(* PLC project PLC411_MAIN, home PLC411_MAIN 1 *)
(* stored: creationDateTime 2019-11-13T09:37:45, productRelease 0, modificationDateTime 2023-05-04T09:24:28, version 0 *)

(* Increment of source value *)
FUNCTION Inc : INT
  VAR_INPUT
    IN : BOOL;  (* execution allow *)
    V : INT;  (* source value *)
  END_VAR
  VAR
    Val : INT;
  END_VAR

            Val:= V;

IF IN = TRUE THEN
  Val:= V+1;
END_IF;

Inc:= Val;


          
END_FUNCTION

(* Decrement of source value *)
FUNCTION Dec : INT
  VAR_INPUT
    IN : BOOL;  (* execution allow *)
    V : INT;  (* source value *)
  END_VAR
  VAR
    Val : INT;
  END_VAR

            Val:= V;

IF IN = TRUE AND Val > 0 THEN
  Val:= V-1;
END_IF;

Dec:= Val;


          
END_FUNCTION

(* Increment of source value (limited) *)
FUNCTION IncLim : INT
  VAR_INPUT
    IN : BOOL;  (* execution allow *)
    V : INT;  (* value *)
    Mn : INT;  (* minimum *)
    Mx : INT;  (* maximum *)
  END_VAR
  VAR
    Val : INT;
  END_VAR

            Val:= Inc(IN:=IN, V:=V);
Val:= LIMIT(MN:=Mn, IN:=Val, MX:=Mx);
IncLim:= Val;
          
END_FUNCTION

(* Decrement of source value (limited) *)
FUNCTION DecLim : INT
  VAR_INPUT
    IN : BOOL;  (* execution allow *)
    V : INT;  (* value *)
    Mn : INT;  (* minimum *)
    Mx : INT;  (* maximum *)
  END_VAR
  VAR
    Val : INT;
  END_VAR

            Val:= Dec(IN:=IN, V:=V);
Val:= LIMIT(MN:=Mn, IN:=Val, MX:=Mx);
DecLim:= Val;
          
END_FUNCTION

(* RAMP-signal (from 0 to 1000) *)
FUNCTION Ramp1000 : WORD
  VAR_INPUT
    IN : BOOL;  (* execution allow *)
    V : WORD;  (* previous RAMP-signal *)
  END_VAR
  VAR
    Val : INT;
  END_VAR

            Val:= WORD_TO_INT(V);

IF IN = TRUE THEN

  Val:= Val+1;
  IF Val >= 1000 THEN
    Val:= 0;
  END_IF;

END_IF;

Ramp1000:= INT_TO_WORD(Val);


          
END_FUNCTION

(* Set bit value in source word *)
FUNCTION SetBitWo : WORD
  VAR_INPUT
    Wo : WORD := 0;  (* source word *)
    Pos : BYTE := 0;  (* bit position (0..15) *)
    Val : BOOL := FALSE;  (* bit value *)
  END_VAR
  VAR
    Mask : WORD := 0;
  END_VAR

            Mask:= REAL_TO_WORD(EXPT(INT_TO_REAL(2),BYTE_TO_INT(Pos)));
IF Val = FALSE THEN
  SetBitWo:= (Wo AND NOT(Mask));
ELSE
  SetBitWo:= (Wo OR Mask);
END_IF;
          
END_FUNCTION

(* 16-bit coder *)
FUNCTION Cd16 : WORD
  VAR_INPUT
    In0 : BOOL := FALSE;  (* value of 0-bit *)
    In1 : BOOL := FALSE;  (* value of 1-bit *)
    In2 : BOOL := FALSE;  (* value of 2-bit *)
    In3 : BOOL := FALSE;  (* value of 3-bit *)
    In4 : BOOL := FALSE;  (* value of 4-bit *)
    In5 : BOOL := FALSE;  (* value of 5-bit *)
    In6 : BOOL := FALSE;  (* value of 6-bit *)
    In7 : BOOL := FALSE;  (* value of 7-bit *)
    In8 : BOOL := FALSE;  (* value of 8-bit *)
    In9 : BOOL := FALSE;  (* value of 9-bit *)
    In10 : BOOL := FALSE;  (* value of 10-bit *)
    In11 : BOOL := FALSE;  (* value of 11-bit *)
    In12 : BOOL := FALSE;  (* value of 12-bit *)
    In13 : BOOL := FALSE;  (* value of 13-bit *)
    In14 : BOOL := FALSE;  (* value of 14-bit *)
    In15 : BOOL := FALSE;  (* value of 15-bit *)
  END_VAR
  VAR
    Val : WORD := 0;
  END_VAR

            Val:= SetBitWo(Wo:=Val, Pos:=INT_TO_BYTE(0), Val:=In0);
Val:= SetBitWo(Wo:=Val, Pos:=INT_TO_BYTE(1), Val:=In1);
Val:= SetBitWo(Wo:=Val, Pos:=INT_TO_BYTE(2), Val:=In2);
Val:= SetBitWo(Wo:=Val, Pos:=INT_TO_BYTE(3), Val:=In3);
Val:= SetBitWo(Wo:=Val, Pos:=INT_TO_BYTE(4), Val:=In4);
Val:= SetBitWo(Wo:=Val, Pos:=INT_TO_BYTE(5), Val:=In5);
Val:= SetBitWo(Wo:=Val, Pos:=INT_TO_BYTE(6), Val:=In6);
Val:= SetBitWo(Wo:=Val, Pos:=INT_TO_BYTE(7), Val:=In7);
Val:= SetBitWo(Wo:=Val, Pos:=INT_TO_BYTE(8), Val:=In8);
Val:= SetBitWo(Wo:=Val, Pos:=INT_TO_BYTE(9), Val:=In9);
Val:= SetBitWo(Wo:=Val, Pos:=INT_TO_BYTE(10), Val:=In10);
Val:= SetBitWo(Wo:=Val, Pos:=INT_TO_BYTE(11), Val:=In11);
Val:= SetBitWo(Wo:=Val, Pos:=INT_TO_BYTE(12), Val:=In12);
Val:= SetBitWo(Wo:=Val, Pos:=INT_TO_BYTE(13), Val:=In13);
Val:= SetBitWo(Wo:=Val, Pos:=INT_TO_BYTE(14), Val:=In14);
Val:= SetBitWo(Wo:=Val, Pos:=INT_TO_BYTE(15), Val:=In15);
Cd16:= Val;

          
END_FUNCTION

(* Get bit value from source word *)
FUNCTION GetBitWo : BOOL
  VAR_INPUT
    Wo : WORD := 0;  (* source word *)
    Pos : BYTE := 0;  (* bit position (0..15) *)
  END_VAR
  VAR
    Mask : WORD := 0;
  END_VAR

            Mask:= REAL_TO_WORD(EXPT(INT_TO_REAL(2),BYTE_TO_INT(Pos)));
GetBitWo:= ((Wo AND Mask) > 0);

          
END_FUNCTION

(* Calculate scale angle factor *)
FUNCTION ScaleA_Ka : REAL
  VAR_INPUT
    Ex : BOOL := FALSE;  (* execution allow *)
    V1 : REAL := 0.0;  (* value of low point *)
    V2 : REAL := 0.0;  (* value of high point *)
    Y1 : REAL := 0.0;  (* calibration value of low point *)
    Y2 : REAL := 0.0;  (* calibration value of high point *)
    Ka : REAL := 0.0;  (* source value of the factor *)
  END_VAR

            IF Ex = TRUE THEN
  ScaleA_Ka:= (Y2-Y1)/(V2-V1);
ELSE  
  ScaleA_Ka:= Ka;
END_IF;

          
END_FUNCTION

(* Calculate scale offset factor *)
FUNCTION ScaleA_Kb : REAL
  VAR_INPUT
    Ex : BOOL := FALSE;  (* execution allow *)
    V1 : REAL := 0.0;  (* value of low point *)
    V2 : REAL := 0.0;  (* value of high point *)
    Y1 : REAL := 0.0;  (* calibration value of low point *)
    Y2 : REAL := 0.0;  (* calibration value of high point *)
    Kb : REAL := 0.0;  (* source value of the factor *)
  END_VAR

            IF Ex = TRUE THEN
  ScaleA_Kb:= ((Y1*V2)-(Y2*V1))/(V2-V1);
ELSE  
  ScaleA_Kb:= Kb;
END_IF;

          
END_FUNCTION

(* Scale of analog value *)
FUNCTION ScaleA : REAL
  VAR_INPUT
    Ex : BOOL := FALSE;  (* execution allow *)
    V : REAL := 0.0;  (* value of curent point *)
    Ka : REAL := 0.0;  (* angle factor *)
    Kb : REAL := 0.0;  (* offset factor *)
    Y : REAL := 0.0;  (* source scale value *)
  END_VAR

            IF Ex = TRUE THEN
  ScaleA:= (Ka*V)+Kb;
ELSE  
  ScaleA:= Y;
END_IF;

          
END_FUNCTION

(* TON Periodical Blink *)
FUNCTION_BLOCK TONb
  VAR_INPUT
    IN : BOOL := FALSE;  (* TON.Start/Stop *)
    PT : TIME := T#0ms;  (* TON.Period *)
  END_VAR
  VAR_OUTPUT
    Q : BOOL := FALSE;  (* TON.BlinkQuit (period for Q = FALSE, pediod for Q=TRUE) *)
    ET : TIME := T#0ms;  (* TON.EstimatedTime *)
  END_VAR
  VAR
    TON0 : TON;
    TON1 : TON;
  END_VAR

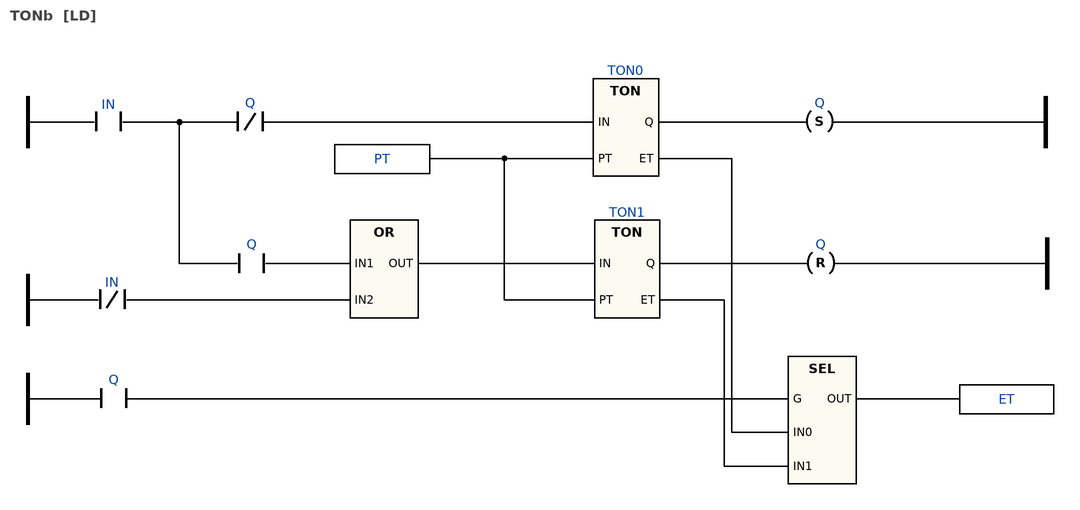
(* LD diagram, written out as Structured Text *)
TON0(IN := IN AND NOT Q, PT := PT);
IF TON0.Q THEN Q := TRUE; END_IF;
TON1(IN := IN AND Q OR NOT IN, PT := PT);
IF TON1.Q THEN Q := FALSE; END_IF;
ET := SEL(Q, TON0.ET, TON1.ET);
END_FUNCTION_BLOCK

(* TON Continuous *)
FUNCTION_BLOCK TONc
  VAR_INPUT
    IN : BOOL := FALSE;  (* start command *)
  END_VAR
  VAR_OUTPUT
    Q : BOOL := FALSE;  (* status *)
    ET : TIME := T#0ms;  (* estimated time *)
  END_VAR
  VAR
    TON1 : TON;
    TON1_IN : BOOL := FALSE;
    TON1_TM : TIME := T#600000ms;
    TON1Inc : TON;
    TON1Inc_IN : BOOL := FALSE;
    TON1Inc_TM : TIME := T#300000ms;
  END_VAR

            TON1_IN   := IN;
TON1Inc_IN:= IN;

IF TON1Inc.Q = TRUE THEN
  TON1_TM   := ADD_TIME(IN1:=TON1_TM, IN2:=TON1Inc_TM);
  TON1Inc_IN:= FALSE;
END_IF;

TON1(IN:=TON1_IN, PT:=TON1_TM);
TON1Inc(IN:=TON1Inc_IN, PT:=TON1Inc_TM);

Q := TON1.Q;
ET:= TON1.ET;

          
END_FUNCTION_BLOCK

(* TON msec *)
FUNCTION_BLOCK TONms
  VAR_INPUT
    IN : BOOL := FALSE;  (* TON.Start/Stop *)
    MS : DWORD := 0;  (* TON.Period (msec) *)
  END_VAR
  VAR_OUTPUT
    Q : BOOL := FALSE;  (* TON.Status (FALSE - counting, TRUE - done) *)
    ET : TIME := T#0ms;  (* TON.EstimatedTime *)
    ETMS : DWORD := 0;  (* TON.EstimatedTime (ms) *)
  END_VAR
  VAR
    TON1 : TON;
    TON1_TM : TIME := T#0ms;
  END_VAR

            IF IN = TRUE THEN
  
  IF MS > 0 THEN
    TON1_TM:= REAL_TO_TIME(DWORD_TO_REAL(MS)/1000.0);
  END_IF;
  
END_IF;

TON1(IN:=IN, PT:=TON1_TM);

IF (MS > 0 AND TON1.Q = TRUE) OR (MS = 0) THEN
  Q:= TRUE;
ELSE
  Q:= FALSE;
END_IF;

ET:= TON1.ET;
ETMS:= REAL_TO_DWORD(TIME_TO_REAL(TON1.ET)*1000.0);

          
END_FUNCTION_BLOCK

(* TON sec *)
FUNCTION_BLOCK TONs
  VAR_INPUT
    IN : BOOL := FALSE;  (* TON.Start/Stop *)
    SEC : WORD := 0;  (* TON.Period (sec) *)
  END_VAR
  VAR_OUTPUT
    Q : BOOL := FALSE;  (* TON.Status (FALSE - counting, TRUE - done) *)
    ET : TIME := T#0ms;  (* TON.EstimatedTime *)
    ETMS : DWORD := 0;  (* TON.EstimatedTime (ms) *)
  END_VAR
  VAR
    TON1 : TON;
    TON1_TM : TIME := T#0ms;
  END_VAR

            IF IN = TRUE THEN
  
  IF SEC > 0 THEN
    TON1_TM:= REAL_TO_TIME(WORD_TO_REAL(SEC));
  END_IF;
  
END_IF;

TON1(IN:=IN, PT:=TON1_TM);

IF (SEC > 0 AND TON1.Q = TRUE) OR (SEC = 0) THEN
  Q:= TRUE;
ELSE
  Q:= FALSE;
END_IF;

ET:= TON1.ET;
ETMS:= REAL_TO_DWORD(TIME_TO_REAL(TON1.ET)*1000.0);

          
END_FUNCTION_BLOCK

(* Filtration of discrete value *)
FUNCTION_BLOCK FiltrD
  VAR_INPUT
    Ex : BOOL := FALSE;  (* execution allow *)
    V : BOOL := FALSE;  (* source value *)
    Tm : TIME := T#0ms;  (* filter delay (ms) *)
  END_VAR
  VAR_OUTPUT
    Ov : BOOL := FALSE;  (* filtered source value *)
  END_VAR
  VAR
    Val : BOOL := FALSE;
    TON0 : TON;
    TON1 : TON;
  END_VAR

            TON0(IN:=AND(Ex, NOT(V)), PT:=Tm);
TON1(IN:=AND(Ex, V), PT:=Tm);

IF TON0.Q = TRUE THEN
  Val:= FALSE;
END_IF;

IF TON1.Q = TRUE THEN
  Val:= TRUE;
END_IF;

Ov:= Val;

          
END_FUNCTION_BLOCK

(* Filtration of analog value *)
FUNCTION_BLOCK FiltrA
  VAR_INPUT
    Ex : BOOL := FALSE;  (* execution allow *)
    V : REAL := 0.0;  (* source value *)
    K : REAL := 0.0;  (* filter factor (0.0 .. 1.0) *)
  END_VAR
  VAR_OUTPUT
    Ov : REAL := 0.0;  (* filtered source value *)
  END_VAR
  VAR
    Val : REAL := 0.0;  (* stored value *)
    Klim : REAL := 0.0;  (* stored value *)
  END_VAR

            IF Ex = TRUE THEN
  Klim:= LIMIT(MN:=0.0, IN:=K, MX:=1.0);
  Val := (Klim*V)+(1.0-Klim)*Ov;
ELSE
  Val:= V;
END_IF;

Ov:= Val;

          
END_FUNCTION_BLOCK

(* 2-Position Regulator *)
FUNCTION_BLOCK Reg2p
  VAR_INPUT
    IN : BOOL := FALSE;  (* Regulator.Start/Stop *)
    V : REAL := 0.0;  (* Process Value *)
    Sp : REAL := 0.0;  (* Setpoint *)
    Hy : REAL := 0.0;  (* Hysteresis (+/- from Sp) for Q.On/Off *)
    Tm : TIME := T#0ms;  (* Output delay *)
  END_VAR
  VAR_OUTPUT
    Q : BOOL := FALSE;  (* Output command *)
  END_VAR
  VAR
    First : BOOL := FALSE;  (* First iteration is completed (TRUE) *)
    TON1 : TON;
    TON1_IN : BOOL := FALSE;
  END_VAR

            IF IN = TRUE THEN
  
  IF (V < Sp AND First = FALSE) OR (V < (Sp-Hy)) THEN
    TON1_IN:= TRUE;
  ELSIF (V > (Sp+Hy)) THEN
    TON1_IN:= FALSE;
  END_IF;

  IF First = FALSE THEN
    First:= TRUE;
  END_IF;
  
ELSE
  First:= FALSE;
  TON1_IN:= FALSE;
  Q:= FALSE;
END_IF;

Q:= TON1.Q;

TON1(IN:=TON1_IN, PT:=Tm);

          
END_FUNCTION_BLOCK

(* Diagnostic of the Control Loop *)
FUNCTION_BLOCK LoopCtrl
  VAR_INPUT
    V : REAL := 0.0;  (* Process Value *)
    CHi : BOOL := FALSE;  (* HighAlarmZone.Allow *)
    DHi : REAL := 0.0;  (* HighAlarmZone.Setpoint *)
    THi : TIME := T#0ms;  (* HighAlarmZone.Delay *)
    CLo : BOOL := FALSE;  (* LowAlarmZone.Allow *)
    DLo : REAL := 0.0;  (* LowAlarmZone.Setpoint *)
    TLo : TIME := T#0ms;  (* LowAlarmZone.Delay *)
  END_VAR
  VAR_OUTPUT
    Q : BOOL := FALSE;  (* Result (TRUE - no breakage, FALSE - breakage) *)
    OK : BYTE := 0;  (* Result code (0 - no breakage, 1 - breakage in Low Zone, 2 - breakage in High Zone) *)
  END_VAR
  VAR
    TON1 : TON;
    TON1_IN : BOOL := FALSE;
    TON1_PT : TIME := T#0ms;
    K : BYTE := 0;  (* Result code (local) *)
  END_VAR

            IF (V < DLo AND CLo = TRUE) THEN
  K:= 1;
  TON1_PT:= TLo;
ELSIF (V > DHi AND CHi = TRUE) THEN
  K:= 2;
  TON1_PT:= THi;
ELSE
  K:= 0;
END_IF;

IF K > 0 THEN
  TON1_IN:= TRUE;
  IF TON1.Q = TRUE THEN
    OK:= K;
  END_IF;
ELSE
  TON1_IN:= FALSE;
  OK:= 0;
END_IF;

TON1(IN:=TON1_IN, PT:=TON1_PT);

IF OK > 0 THEN
  Q:= TRUE;
ELSE
  Q:= FALSE;
END_IF;

          
END_FUNCTION_BLOCK

(* PID-controller (v1) *)
FUNCTION_BLOCK PID1
  VAR_INPUT
    Ex : BOOL := FALSE;  (* execution allow *)
    V : REAL := 0.0;  (* source value *)
    Sp : REAL := 0.0;  (* setpoint *)
    Ty : BYTE := 0;  (* type of controller *)
    Pro : BYTE := 0;  (* type of process *)
    Kp : REAL := 0.0;  (* P-factor *)
    Ki : REAL := 0.0;  (* I-factor *)
    Kd : REAL := 0.0;  (* D-factor *)
    Sck : BOOL := FALSE;  (* external command to start regulator cycle *)
    dI : REAL := 0.0;  (* integral zone *)
    dZ : REAL := 0.0;  (* dead zone *)
    Ym : BYTE := 0;  (* type of OY *)
  END_VAR
  VAR_OUTPUT
    Ok : BYTE := 0;  (* result code *)
    OY : REAL := 0.0;  (* regulator value (%) *)
  END_VAR
  VAR
    Er : REAL := 0.0;  (* error delta *)
    ErAbs : REAL := 0.0;  (* error delta (absolute) *)
    ErPrev : REAL := 0.0;  (* error delta (previous cycle) *)
    ErDiff : REAL := 0.0;  (* error delta (diff) *)
    Ppart : REAL := 0.0;  (* P-part *)
    Ipart : REAL := 0.0;  (* I-part *)
    Dpart : REAL := 0.0;  (* D-part *)
    SckSet : BOOL := FALSE;  (* external start (set) *)
    ErrorSet : BOOL := FALSE;  (* e-zone (set) *)
  END_VAR

            (* Ty - regulator type *)
(* = 0 - PID *)
(* = 1 - PI *)
(* = 2 - PD *)
(* = 3 - P *)

(* Pro - process type *)
(* = 0 - increasing (by default) *)
(* = 1 - decreasing *)

(* Ym - type of OY *)
(* = 0 - unipolar    0.0 .. 100.0 % (by default) *)
(* = 1 - bipolar  -100.0 .. 100.0 % *)

(* Ok - result code *)
(* = 0 - work *)
(* = 1 - off *)
(* = 2 - dead (d-)zone *)
(* = 3 - integral (i-)zone *)
(* = 4 - incorrect regulator type *)

(* reset Sck *)
IF Sck = FALSE THEN
  SckSet:= FALSE;
END_IF;

(* test execution allow *)
IF Ex = TRUE THEN
  
  (* test regulator type *)
  IF Ty <= 3 THEN
    
    (* test start *)
    IF Sck = TRUE AND SckSet = FALSE AND ErrorSet = FALSE THEN
      
      SckSet:= TRUE;
      
      (* work *)
      Ok:= 0;
     
      Er    := (Sp-V);
      ErDiff:= (Er-ErPrev);
      ErPrev:= Er;
      ErAbs := ABS(IN:=Er);
      
      (* test d-zone *)
      IF ErAbs >= dZ THEN
        
        (* Ty: 0-PID, 1-PI, 2-PD, 3-P *)
        Ppart:= (Kp*Er);
        
        (* Ty: 0-PID, 1-PI *)
        IF (Ty = 0 OR Ty = 1) AND (ErAbs < dI OR dI = 0.0) AND Ki > 0.0 THEN
          (* i-zone *)
          Ok:= 3;
          Ipart:= (Ipart+Er);
          IF Ipart >= Ki THEN
            Ipart:= Ki;
          END_IF;
          Ipart:= ((1.0/Ki)*Ipart);
        ELSE
          Ipart:= 0.0;
        END_IF;
        
        (*0-PID, 2-PD*)
        IF (Ty = 0 OR Ty = 2) THEN
          Dpart:= (Kd*ErDiff);
        ELSE
          Dpart:= 0.0;
        END_IF;
        
        OY:= (Ppart+Ipart+Dpart)*100.0;
        
      ELSE
        (* d-zone *)
        Ok:= 2;
      END_IF;
      (* end of test d-zone *)
      
    END_IF;
    (* end of test start *)
  
  ELSE
    (* incorrect regulator type *)
    Ok:= 4;
    ErrorSet:= TRUE;
  END_IF;
  (* end of test regulator type *)
  
ELSE
  (* off *)
  Ok:= 1;
END_IF;
(* end of Ex *) 

(* off *)
IF Ok = 1 THEN
  OY       := 0.0;
  SckSet   := FALSE;
  ErrorSet := FALSE;
  Ppart    := 0.0;
  Ipart    := 0.0;
  Dpart    := 0.0;
END_IF;

(* error of regulator type *)
IF ErrorSet = TRUE THEN
  OY       := 0.0;
END_IF;

(* scale OY by type of process *)
IF Pro = 1 THEN
  (* decreasing *)
  OY:= (100.0-OY);
END_IF;

(* scale OY by type of output *)
IF Ym = 1 THEN
  (* bipolar *)
  OY:= LIMIT(MN:=-100.0, IN:=OY, MX:=100.0);
ELSE
  (* unipolar *)
  OY:= LIMIT(MN:=0.0, IN:=OY, MX:=100.0);
END_IF;

          
END_FUNCTION_BLOCK

(* PID-controller (v2) *)
FUNCTION_BLOCK PID2
  VAR_INPUT
    Ex : BOOL := FALSE;  (* execution allow *)
    V : REAL := 0.0;  (* source value *)
    Sp : REAL := 0.0;  (* setpoint *)
    Ty : BYTE := 0;  (* type of controller *)
    Pro : BYTE := 0;  (* type of process *)
    Kp : REAL := 0.0;  (* P-factor *)
    Ki : REAL := 0.0;  (* I-factor *)
    Kd : REAL := 0.0;  (* D-factor *)
    Tm : DWORD := 1000;  (* cycle time (ms) *)
    dI : REAL := 0.0;  (* integral zone *)
    dZ : REAL := 0.0;  (* dead zone *)
    Ym : BYTE := 0;  (* type of OY *)
  END_VAR
  VAR_OUTPUT
    Ok : BYTE := 0;  (* result code *)
    OY : REAL := 0.0;  (* regulator value (%) *)
  END_VAR
  VAR
    TON_Work : TON;
    TON_Work_IN : BOOL := FALSE;
    TON_Work_TM : TIME := T#0ms;
    PID1_1 : PID1;
  END_VAR

            PID1_1(Ex:=Ex, V:=V, Sp:=Sp, Ty:=Ty, Pro:=Pro, Kp:=Kp, Ki:=Ki, Kd:=Kd, Sck:=TON_Work.Q, dI:=dI, dZ:=dZ, Ym:=Ym);

Ok:= PID1_1.Ok;
OY:= PID1_1.OY;

IF Ex = TRUE AND Tm > 0 THEN
  TON_Work_TM:= REAL_TO_TIME(DWORD_TO_REAL(Tm)/1000.0);
  TON_Work_IN:= TRUE;
ELSE
  TON_Work_IN:= FALSE;
END_IF;

IF TON_Work.Q = TRUE THEN
  TON_Work_IN:= FALSE;
END_IF;

TON_Work(IN:=TON_Work_IN, PT:=TON_Work_TM);

(* DEBUG *)
(* set Class of debug variables to Output to use its as Outputs of the FB *)
(* set Class of debug variables to Local to hide its *)
(* Deb_P   := PID1_1.Deb_P; *)
(* Deb_I   := PID1_1.Deb_I; *)
(* Deb_D   := PID1_1.Deb_D; *)
(* Deb_Et  := REAL_TO_DWORD(TIME_TO_REAL(TON_Work.ET)*1000.0); *)
(* Deb_dEEt:= PID1_1.Deb_dEEt; *)
(* end of DEBUG *)

          
END_FUNCTION_BLOCK

(* Autotuning of PID-controller *)
FUNCTION_BLOCK PIDtun
  VAR_INPUT
    Ex : BOOL := FALSE;  (* execution allow *)
    V : REAL := 0.0;  (* source value *)
    Diff : REAL := 0.0;  (* difference setpoint *)
    Ty : BYTE := 0;  (* type of controller *)
    Pro : BYTE := 0;  (* type of process *)
  END_VAR
  VAR_OUTPUT
    Ok : BYTE := 0;  (* result code *)
    OY : REAL := 0.0;  (* regulator value *)
    OKp : REAL := 0.0;  (* P-factor *)
    OKi : REAL := 0.0;  (* I-factor *)
    OKd : REAL := 0.0;  (* D-factor *)
    OTm : DWORD := 0;  (* cycle time (ms) *)
  END_VAR
  VAR
    TunDone : BOOL := FALSE;
    Tm1 : REAL := 0.0;  (* t0 (ms) *)
    Tm2 : REAL := 0.0;  (* tu (ms) *)
    TmSum : REAL := 0.0;  (* t (ms) *)
    V1Set : BOOL := FALSE;
    V01 : REAL := 0.0;
    V063 : REAL := 0.0;
    Rr : REAL := 0.0;  (* R *)
    Tm1sec : REAL := 0.0;  (* t0 div 100 *)
    TONcont1 : TONc;
    TONcont1_IN : BOOL := FALSE;
  END_VAR

            (* Ty - regulator type *)
(* = 0 - PID *)
(* = 1 - PI *)
(* = 2 - PD *)
(* = 3 - P *)

(* Pro - process type *)
(* = 0 - increasing (by default) *)
(* = 1 - decreasing *)

(* Ok - result code *)
(* = 0 - work *)
(* = 1 - off *)
(* = 2 - incorrect regulator type *)
(* = 3 - work done success *)

IF Ex = TRUE THEN
  
  IF Ty <= 3 THEN
      
    IF TunDone = FALSE THEN
      
      (* work *)
      Ok:= 0;
      
      IF V1Set = FALSE THEN
        V1Set:= TRUE;
        (* calculate setpoint for V(0.1) by type of process *)
        IF Pro = 1 THEN
          (* decreasing *)
          V01 := (V-(0.1*Diff));
          V063:= (V-(0.63*Diff));
        ELSE
          (* increasing *)
          V01 := (V+(0.1*Diff));
          V063:= (V+(0.63*Diff));
        END_IF;
      END_IF;
      
      (* set Tm1 (ms) *)
      IF V < V01 THEN
        Tm1:= TIME_TO_REAL(TONcont1.ET)*1000.0;
      END_IF;
      
      (* set Tm2 (ms) *)
      IF V >= V063 THEN
        
        TONcont1_IN:= FALSE;
        TunDone    := TRUE;
        
        Tm2   := TIME_TO_REAL(TONcont1.ET)*1000.0;
        TmSum := (Tm1+Tm2);
        OTm   := REAL_TO_DWORD((Tm1*1.875));
        Rr    := (Diff/((TmSum-Tm1)/1000.0));
        Tm1sec:= (Tm1/1000.0);
        (* 1000 - divider to convert msec to sec *)
          
        (* calculate factors by type of regulator *)
        CASE BYTE_TO_INT(Ty) OF
          0:
            (* PID *)
            OKp:= (1.2/(Rr*Tm1sec));
            OKi:= (2.0*Tm1sec);
            OKd:= (0.4*Tm1sec);
          1:
            (* PI *)
            OKp:= (0.8/(Rr*Tm1sec));
            OKi:= (2.0*Tm1sec);
          2:
            (*PD*)
            OKp:= (1.0/(Rr*Tm1sec));
            OKd:= (0.25*Tm1sec);
          3:
            (*P*)
            OKp:= (1.0/(Rr*Tm1sec));
        END_CASE;
        
      END_IF;
      (* end of Tm2 *)
    ELSE
      (* work done success *)
      Ok:= 3;
    END_IF;
    (* end of TunDone *)
  ELSE
    (* incorrect regulator type *)
    Ok:= 2;
  END_IF;
  (* end of Ty *)
ELSE
  (* off *)
  Ok:= 1;
END_IF;
(* end of Ex *)

(* work *)
IF Ok = 0 THEN
  OY         := 100.0;
  TONcont1_IN:= TRUE;
END_IF;

(* off, error *)
IF Ok = 1 OR Ok = 2 THEN
  OY         := 0.0;
  TONcont1_IN:= FALSE;
  V1Set      := FALSE;
  TunDone    := FALSE;
  OKp        := 0.0;
  OKi        := 0.0;
  OKd        := 0.0;
  OTm        := 0;
END_IF;

(* work is done success *)
IF TunDone = TRUE THEN
  OY         := 0.0;
END_IF;

TONcont1(IN:=TONcont1_IN);

(* DEBUG *)
(* set Class of debug variables to Output to use its as Outputs of the FB *)
(* set Class of debug variables to Local to hide its *)
(* Deb_V1 := V01; *)
(* Deb_Tm1:= Tm1; *)
(* Deb_V2 := V063; *)
(* Deb_Tm2:= Tm2; *)
(* end of DEBUG *)

          
END_FUNCTION_BLOCK

(* FuzzyLogic-controller (v1) *)
FUNCTION_BLOCK FLR1
  VAR_INPUT
    Ex : BOOL := FALSE;  (* execution allow *)
    V : REAL := 0.0;  (* source value *)
    Sp : REAL := 0.0;  (* setpoint *)
    Pro : BYTE := 0;  (* type of process *)
    Sck : BOOL := FALSE;  (* external command to start regulator cycle *)
    Tm : DWORD := 0;  (* cycle time (ms) *)
    dV : REAL := 0.0;  (* increment step of OY (%) *)
    dZ : REAL := 0.0;  (* dead zone *)
    Ym : BYTE := 0;  (* type of OY *)
  END_VAR
  VAR_OUTPUT
    Ok : BYTE := 0;  (* result code *)
    OY : REAL := 0.0;  (* regulator value (%) *)
  END_VAR
  VAR
    Vprev : REAL := 0.0;  (* previous source value *)
    TmDv : REAL := 0.0;  (* dV time (ms) *)
    UpDown : SINT := 0;  (* flag UpDown *)
    SckSet : BOOL := FALSE;  (* external start (set) *)
    ErrorSet : BOOL := FALSE;  (* e-zone (set) *)
    Er : REAL := 0.0;  (* error delta *)
    TON_Dv : TON;
    TON_Dv_IN : BOOL := FALSE;
    TON_Dv_TM : TIME := T#0ms;
  END_VAR

            (* Pro - process type *)
(* = 0 - increasing (by default) *)
(* = 1 - decreasing *)

(* Ym - type of OY *)
(* = 0 - unipolar    0.0 .. 100.0 % (by default) *)
(* = 1 - bipolar  -100.0 .. 100.0 % *)

(* Ok - result code *)
(* = 0 - work *)
(* = 1 - off *)
(* = 2 - dead (d-)zone *)
(* = 4 - control failure (e-)zone *)

(* reset Sck *)
IF Sck = FALSE THEN
  SckSet:= FALSE;
END_IF;

(* test execution allow *)
IF Ex = TRUE THEN
    
  (* test start *)
  IF Sck = TRUE AND SckSet = FALSE AND ErrorSet = FALSE THEN
    
    SckSet:= TRUE;  
          
    (* work *)
    Ok:= 0;
    
    Er:= (Sp-V);
    
    (* test d-zone *)
    IF ABS(IN:=Er) >= dZ THEN
      (* exec *)
      {extern void AppFlr(FLR1*);AppFlr(data__);}
    ELSE
      (* d-zone *)
      Ok:= 2;
    END_IF;
    (* end of test d-zone *)
      
  END_IF;
  (* end of test start *)
  
ELSE
  (* off *)
  Ok:= 1;
END_IF;
(* end of Ex *) 

(* work *)
IF Ok = 0 THEN
  
  IF TmDv > 0.0 THEN
    (* msec to real-sec to time *)
    TON_Dv_TM:= REAL_TO_TIME(TmDv/1000.0);
    TON_Dv_IN:= TRUE;
  END_IF;
  
  IF TON_Dv.Q = TRUE THEN
    TON_Dv_IN:= FALSE;
    (* down *)
    IF UpDown = -1 THEN
      OY:= OY-dV;
    END_IF;
    (* up *)
    IF UpDown = 1 THEN
      OY:= OY+dV;
    END_IF;
  END_IF;
  
ELSE
  TON_Dv_IN:= FALSE;
END_IF;
(* end of work *)


(* off *)
IF Ok = 1 THEN
  OY       := 0.0;
  SckSet   := FALSE;
  ErrorSet := FALSE;
  Vprev    := 0.0;
END_IF;

(* error *)
IF ErrorSet = TRUE THEN
  OY       := 0.0;
END_IF;

(* scale OY by type of process *)
IF Pro = 1 THEN
  (* decreasing *)
  OY:= (100.0-OY);
END_IF;

(* scale OY by type of output *)
IF Ym = 1 THEN
  (* bipolar *)
  OY:= LIMIT(MN:=-100.0, IN:=OY, MX:=100.0);
ELSE
  (* unipolar *)
  OY:= LIMIT(MN:=0.0, IN:=OY, MX:=100.0);
END_IF;

TON_Dv(IN:=TON_Dv_IN, PT:=TON_Dv_TM);

          
END_FUNCTION_BLOCK

(* FuzzyLogic-controller (v2) *)
FUNCTION_BLOCK FLR2
  VAR_INPUT
    Ex : BOOL := FALSE;  (* execution allow *)
    V : REAL := 0.0;  (* source value *)
    Sp : REAL := 0.0;  (* setpoint *)
    Pro : BYTE := 0;  (* type of process *)
    Tm : DWORD := 0;  (* cycle time (ms) *)
    dV : REAL := 0.0;  (* increment step of OY (%) *)
    dZ : REAL := 0.0;  (* dead zone *)
    Ym : BYTE := 0;  (* type of OY *)
  END_VAR
  VAR_OUTPUT
    Ok : BYTE := 0;  (* result code *)
    OY : REAL := 0.0;  (* regulator value (%) *)
  END_VAR
  VAR
    TON_Work : TON;
    TON_Work_IN : BOOL := FALSE;
    TON_Work_TM : TIME := T#0ms;
    FLR1_1 : FLR1;
  END_VAR

            FLR1_1(Ex:=Ex, V:=V, Sp:=Sp, Pro:=Pro, Sck:=TON_Work.Q, Tm:=Tm, dV:=dV, dZ:=dZ, Ym:=Ym);

Ok:= FLR1_1.Ok;
OY:= FLR1_1.OY;

IF Ex = TRUE AND Tm > 0 THEN
  (* msec to real-sec to time *)
  TON_Work_TM:= REAL_TO_TIME(DWORD_TO_REAL(Tm)/1000.0);
  TON_Work_IN:= TRUE;
ELSE
  TON_Work_IN:= FALSE;
END_IF;

IF TON_Work.Q = TRUE THEN
  TON_Work_IN:= FALSE;
END_IF;

TON_Work(IN:=TON_Work_IN, PT:=TON_Work_TM);

(* DEBUG *)
(* set Class of debug variables to Output to use its as Outputs of the FB *)
(* set Class of debug variables to Local to hide its *)
(* Deb_Speed := FLR1_1.Deb_Speed; *)
(* Deb_UpDown:= FLR1_1.Deb_UpDown; *)
(* Deb_dVTm  := FLR1_1.Deb_dVTm; *)
(* Deb_dVEt  := FLR1_1.Deb_dVEt; *)
(* Deb_dEEt  := FLR1_1.Deb_dEEt; *)
(* Deb_Et    := REAL_TO_DWORD(TIME_TO_REAL(TON_Work.ET)*1000.0); *)
(* Deb_Y0    := FLR1_1.Deb_Y0; *)
(* Deb_Er    := FLR1_1.Deb_Er; *)
(* Deb_Cm    := FLR1_1.Deb_Cm; *)
(* Deb_m     := FLR1_1.Deb_m; *)
(* end of DEBUG *)

          
END_FUNCTION_BLOCK

(* Autotuning of FLR-controller *)
FUNCTION_BLOCK FLRtun
  VAR_INPUT
    Ex : BOOL := FALSE;  (* execution allow *)
    V : REAL := 0.0;  (* source value *)
    Diff : REAL := 0.0;  (* difference setpoint *)
    Pro : BYTE := 0;  (* type of process *)
  END_VAR
  VAR_OUTPUT
    Ok : BYTE := 0;  (* result code *)
    OY : REAL := 0.0;  (* regulator value *)
    OTm : DWORD := 0;  (* cycle time (ms) *)
  END_VAR
  VAR
    TunDone : BOOL := FALSE;
    Tm1 : REAL := 0.0;  (* t0 (ms) *)
    V1Set : BOOL := FALSE;
    V01 : REAL := 0.0;
    TONcont1 : TONc;
    TONcont1_IN : BOOL := FALSE;
  END_VAR

            (* Pro - process type *)
(* = 0 - increasing (by default) *)
(* = 1 - decreasing *)

(* Ok - result code *)
(* = 0 - work *)
(* = 1 - off *)
(* = 3 - work done success *)

IF Ex = TRUE THEN
  
  IF TunDone = FALSE THEN
      
    (* work *)
    Ok:= 0;
      
    IF V1Set = FALSE THEN
      V1Set:= TRUE;
      (* calculate setpoint for V(0.1) by type of process *)
      IF Pro = 1 THEN
        (* decreasing *)
        V01 := (V-(0.1*Diff));
      ELSE
        (* increasing *)
        V01 := (V+(0.1*Diff));
      END_IF;
    END_IF;
      
    (* set Tm1 (ms) *)
    IF V < V01 THEN
      Tm1:= TIME_TO_REAL(TONcont1.ET)*1000.0;
    ELSE
      OTm:= REAL_TO_DWORD((Tm1*1.875));
      TunDone:= TRUE;
      (* work done success *)
      Ok:= 3;
    END_IF;
    
  END_IF;
  (* end of TunDone *)
    
ELSE
  (* off *)
  Ok:= 1;
END_IF;
(* end of Ex *)

(* work *)
IF Ok = 0 THEN
  OY         := 100.0;
  TONcont1_IN:= TRUE;
END_IF;

(* off, error *)
IF Ok = 1 THEN
  OY         := 0.0;
  TONcont1_IN:= FALSE;
  V1Set      := FALSE;
  TunDone    := FALSE;
  OTm        := 0;
END_IF;

(* work is done success *)
IF TunDone = TRUE THEN
  OY         := 0.0;
  TONcont1_IN:= FALSE;
END_IF;

TONcont1(IN:=TONcont1_IN);

(* DEBUG *)
(* set Class of debug variables to Output to use its as Outputs of the FB *)
(* set Class of debug variables to Local to hide its *)
(* Deb_V1 := V01; *)
(* Deb_Tm1:= Tm1; *)
(* end of DEBUG *)

          
END_FUNCTION_BLOCK

(* 16-bit decoder *)
FUNCTION_BLOCK Dc16
  VAR_INPUT
    V : WORD := 0;  (* Value (bitfield) *)
  END_VAR
  VAR_OUTPUT
    O0 : BOOL := FALSE;  (* Value of 0-bit *)
    O1 : BOOL := FALSE;  (* Value of 1-bit *)
    O2 : BOOL := FALSE;  (* Value of 2-bit *)
    O3 : BOOL := FALSE;  (* Value of 3-bit *)
    O4 : BOOL := FALSE;  (* Value of 4-bit *)
    O5 : BOOL := FALSE;  (* Value of 5-bit *)
    O6 : BOOL := FALSE;  (* Value of 6-bit *)
    O7 : BOOL := FALSE;  (* Value of 7-bit *)
    O8 : BOOL := FALSE;  (* Value of 8-bit *)
    O9 : BOOL := FALSE;  (* Value of 9-bit *)
    O10 : BOOL := FALSE;  (* Value of 10-bit *)
    O11 : BOOL := FALSE;  (* Value of 11-bit *)
    O12 : BOOL := FALSE;  (* Value of 12-bit *)
    O13 : BOOL := FALSE;  (* Value of 13-bit *)
    O14 : BOOL := FALSE;  (* Value of 14-bit *)
    O15 : BOOL := FALSE;  (* Value of 15-bit *)
  END_VAR

            O0 := GetBitWo(Wo:=V, Pos:=INT_TO_BYTE(0));
O1 := GetBitWo(Wo:=V, Pos:=INT_TO_BYTE(1));
O2 := GetBitWo(Wo:=V, Pos:=INT_TO_BYTE(2));
O3 := GetBitWo(Wo:=V, Pos:=INT_TO_BYTE(3));
O4 := GetBitWo(Wo:=V, Pos:=INT_TO_BYTE(4));
O5 := GetBitWo(Wo:=V, Pos:=INT_TO_BYTE(5));
O6 := GetBitWo(Wo:=V, Pos:=INT_TO_BYTE(6));
O7 := GetBitWo(Wo:=V, Pos:=INT_TO_BYTE(7));
O8 := GetBitWo(Wo:=V, Pos:=INT_TO_BYTE(8));
O9 := GetBitWo(Wo:=V, Pos:=INT_TO_BYTE(9));
O10:= GetBitWo(Wo:=V, Pos:=INT_TO_BYTE(10));
O11:= GetBitWo(Wo:=V, Pos:=INT_TO_BYTE(11));
O12:= GetBitWo(Wo:=V, Pos:=INT_TO_BYTE(12));
O13:= GetBitWo(Wo:=V, Pos:=INT_TO_BYTE(13));
O14:= GetBitWo(Wo:=V, Pos:=INT_TO_BYTE(14));
O15:= GetBitWo(Wo:=V, Pos:=INT_TO_BYTE(15));

          
END_FUNCTION_BLOCK

(* Convert msec to TIME *)
FUNCTION MsecToTime : TIME
  VAR_INPUT
    MS : DWORD := 0;  (* msec *)
  END_VAR

            MsecToTime:= REAL_TO_TIME(DWORD_TO_REAL(MS)/1000.0);

          
END_FUNCTION

(* Convert sec to TIME *)
FUNCTION SecToTime : TIME
  VAR_INPUT
    SEC : WORD := 0;  (* sec *)
  END_VAR

            SecToTime:= REAL_TO_TIME(WORD_TO_REAL(SEC));

          
END_FUNCTION
